PROGRAM PRG_TXI_VAC_PUMPS
VAR
    dummy_gauge : ST_VG;
END_VAR

//beamline dummy gauge
dummy_gauge.xPRESS_OK := TRUE;
dummy_gauge.xAT_VAC := TRUE;
dummy_gauge.eState := ValidLo;
dummy_gauge.rPRESS := 1e-4;

//B940-009-R17-PCI-03
fb_PC2L1_L2SI_PIP_01(i_stGauge := dummy_gauge, i_xOverrideMode := xSystemOverrideMode1);
fb_ST1L1_PPS_PIP_01(i_stGauge := fb_ST1L1_PPS_GPI_01.PG, i_xOverrideMode := xSystemOverrideMode1);
fb_TV2L1_PLEG_PIP_01(i_stGauge := fb_TV2L1_PLEG_GPI_01.PG, i_xOverrideMode := xSystemOverrideMode1);
fb_TV3L1_PLEG_PIP_01(i_stGauge := fb_TV2L1_PLEG_GPI_01.PG, i_xOverrideMode := xSystemOverrideMode1);

//B940-009-R17-PCI-04
fb_TV4L1_PLEG_PIP_01(i_stGauge := fb_TV4L1_PLEG_GPI_01.PG, i_xOverrideMode := xSystemOverrideMode1);

END_PROGRAM

(* stored: Version 1.1.0.1, ProductVersion 3.1.4024.6
   POU PRG_TXI_VAC_PUMPS: Id {3fa39cc4-d092-48cb-adaa-6e39f89b2e24}, SpecialFunc None *)
